FUNCTION_BLOCK LINKEVENTRECEIVER (* Service Interface Function Block Type *)
  (* Standard: 61499-2 *)
  (* Version 0.0, 9/14/2008, Horst Mayer, nxtControl GmbH, template *)
  PACKAGE IEC61499;
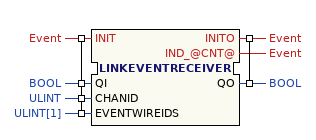
  EVENT_INPUT
    INIT WITH QI, CHANID, EVENTWIREIDS;
  END_EVENT
  EVENT_OUTPUT
    INITO WITH QO;
    IND_@CNT@;
  END_EVENT
  VAR_INPUT
    QI : BOOL;
    CHANID : ULINT;
    EVENTWIREIDS : ARRAY [0..0] OF ULINT;
  END_VAR
  VAR_OUTPUT
    QO : BOOL; (* Event Output Qualifier *)
  END_VAR
END_FUNCTION_BLOCK
